{attribute 'GeneratedUsingTerminal: EL2535-0000-0016'}
{attribute addProperty BoxType "EL2535-0000-0016"}
{attribute addProperty Id "PWM_Status_Channel_1AT %I*PWM_Status_Channel_2D1AF3405PWM_Status_Channel_2AT %I*PWM_Status_Channel_2D1AF3405PWM_Control_Channel_1AT %Q*PWM_Control_Channel_63F162E45PWM_Control_Channel_2AT %Q*PWM_Control_Channel_63F162E45WcStateAT %I*WcState_9091E0EB2InfoDataAT %I*InfoData_32EB74EA10"}
{attribute addProperty CRC "1329227671"}
{attribute addProperty Size "32"}
TYPE EL2535_4F3A6797 EXTENDS EtcSlaveTerminalBase_947E5A46 :
STRUCT
	{attribute addProperty Name "PWM_Status_Channel_1"}
	PWM_Status_Channel_1 : PWM_Status_Channel_2D1AF340;
	{attribute addProperty Name "PWM_Status_Channel_2"}
	PWM_Status_Channel_2 : PWM_Status_Channel_2D1AF340;
	{attribute addProperty Name "PWM_Control_Channel_1"}
	PWM_Control_Channel_1 : PWM_Control_Channel_63F162E4;
	{attribute addProperty Name "PWM_Control_Channel_2"}
	PWM_Control_Channel_2 : PWM_Control_Channel_63F162E4;
	{attribute addProperty Name "WcState"}
	WcState : WcState_9091E0EB;
	{attribute addProperty Name "InfoData"}
	InfoData : InfoData_32EB74EA;
END_STRUCT
END_TYPE

(* stored: Version 1.2.0.0, ProductVersion 3.1.4024.9
   DUT EL2535_4F3A6797: Id {4c9c1933-9dd1-4748-a934-030115e6b5e7} *)
